PROGRAM MAIN
VAR
	i: INT;
	
	nState: INT;
	fbReceiveData: ReceiveData;
	aReceiveData: ARRAY[1..6] OF BYTE;
	aSuffixData: ARRAY[1..2] OF BYTE := [13, 10];
	sDeviceId: STRING(80);
	
	nCursor: INT := 1;
	nRegconizedDeviceIds: INT;
	nTotalDevices: INT;
	aNullId: ARRAY[1..4] OF BYTE;
	aDeviceCount: ARRAY[1..10] OF ST_DeviceCount;
END_VAR

CASE nState OF
	0: // Check if any data is received
		IF GVL.RxBuffer.Count <> 0 THEN
			nState := nState + 1;
		END_IF
	1: // Receive data
		fbReceiveData(
			pPrefix:= , 
			LenPrefix:= , 
			pSuffix:= ADR(aSuffixData), 
			LenSuffix:= 2, 
			pReceiveData:= ADR(aReceiveData), 
			SizeReceiveData:= 6, 
			Timeout:= T#1S, 
			Reset:= , 
			DataReceived=> , 
			busy=> , 
			Error=> , 
			RxTimeout=> , 
			LenReceiveData=> , 
			RXbuffer:= GVL.RxBuffer);
		IF NOT fbReceiveData.busy THEN
			IF fbReceiveData.Error <> 0 THEN
				nState := 100;
			ELSE
				IF fbReceiveData.LenReceiveData = 6 THEN
					nState := nState + 1;
				END_IF
			END_IF
		END_IF
	2: // Get the barcode and check whether it was regconized
		sDeviceId := '';
		FOR i := 1 TO 4 DO
			sDeviceId := CONCAT(sDeviceId, CHR(aReceiveData[i]));
		END_FOR
		nState := 3;		
		FOR i := 1 TO 10 DO
			IF MEMCMP(ADR(aDeviceCount[i].aId), ADR(aReceiveData), 4) = 0 THEN
				nState := 4;
				EXIT;
			END_IF
		END_FOR
	3: // Realize the received barcode as a new barcode which was not known before
		IF nCursor < 11 THEN
			MEMCPY(ADR(aDeviceCount[nCursor].aId), ADR(aReceiveData), 4);
			nRegconizedDeviceIds := nRegconizedDeviceIds + 1;
			nCursor := nCursor + 1;
			nState := nState + 1;
		ELSE
			nState := 100;		
		END_IF
	4: // Increase the number of time the received bar code read
		FOR i := 1 TO 10 DO
			IF MEMCMP(ADR(aDeviceCount[i].aId), ADR(aReceiveData), 4) = 0 THEN
				aDeviceCount[i].nCount := aDeviceCount[i].nCount + 1;
				EXIT;
			END_IF
		END_FOR
		nTotalDevices := nTotalDevices + 1;
		nState := 0;
END_CASE

END_PROGRAM

(* stored: Version 1.1.0.1, ProductVersion 3.1.4024.11
   POU MAIN: Id {2b30c86f-c39a-4e51-8d34-0affd763fdf3}, SpecialFunc None *)
